// TIA Portal V20 export
DATA_BLOCK "DB_PartManagement"   // DB87
// stored: InstanceOfName FB_PartManagement, InstanceOfType FB
"FB_PartManagement"
   // VAR
   //    sShuttle1DrilledPart : "FB_StatusPart";
   //    sShuttle1UndrilledPart { S7_SetPoint := 'True'} : "FB_StatusPart";
   //    sShuttle2DrilledPart { S7_SetPoint := 'True'} : "FB_StatusPart";
   //    sShuttle2UndrilledPart { S7_SetPoint := 'True'} : "FB_StatusPart";
   //    sShuttle1DrilledBw : "FB_StatusPart";
   //    sShuttle1UndrilledBw { S7_SetPoint := 'True'} : "FB_StatusPart";
   //    sShuttle2DrilledBw { S7_SetPoint := 'True'} : "FB_StatusPart";
   //    sShuttle2UndrilledBw { S7_SetPoint := 'True'} : "FB_StatusPart";
   //    sGripperDrilledPart : "FB_StatusPart";
   //    sGripperUndrilledPart { S7_SetPoint := 'True'} : "FB_StatusPart";
   //    sGripperDrilledBw : "FB_StatusPart";
   //    sGripperUndrilledBw { S7_SetPoint := 'True'} : "FB_StatusPart";
   //    sFixtureDrilledPart : "FB_StatusPart";
   //    sFixtureUndrilledPart { S7_SetPoint := 'True'} : "FB_StatusPart";
   //    sFixtureDrilledBw : "FB_StatusPart";
   //    sFixtureUndrilledBw { S7_SetPoint := 'True'} : "FB_StatusPart";
   //    sPosition { S7_SetPoint := 'True'} : "FB_Position";
   // END_VAR
BEGIN
END_DATA_BLOCK
